(* CoDeSys 2.3.9.37 project: Cap5_2.pro *)
(* Libraries: Standard.lib 4.10.05 12:14:46 *)

(* POU PLC_PRG, ST *)
PROGRAM PLC_PRG
VAR
  cont:INT;
	valor1: INT;
	valor2: INT;
      instanciaFB:suma1FB;
END_VAR
valor1:=suma1();
instanciaFB(salidaFB=>valor2);
END_PROGRAM

(* POU suma1FB, ST *)
FUNCTION_BLOCK suma1FB
VAR_INPUT
END_VAR
VAR_OUTPUT
 salidaFB:INT;
END_VAR
VAR
	contador:INT :=0 ;
END_VAR
contador:=contador+1;
salidaFB:=contador;
END_FUNCTION_BLOCK

(* POU suma1, ST *)
FUNCTION suma1 : INT
VAR_INPUT
END_VAR
VAR
  contador:INT :=0;
END_VAR
contador:=contador+1;
suma1:=contador;
END_FUNCTION
